FUNCTION F_CheckDivInt : INT
VAR_INPUT
	divisor: INT;
END_VAR

IF divisor = 0 THEN
	F_CheckDivInt:=1;
ELSE
	F_CheckDivInt:=divisor;
END_IF;

END_FUNCTION

(* stored: Version 1.1.0.1, ProductVersion 3.1.4022.6
   POU F_CheckDivInt: Id {36e81023-df22-4a76-8017-92a1a7b6adaf}, SpecialFunc None *)
